// TIA Portal V19 export
FUNCTION_BLOCK "TYPIC_C215_SF_PBK"   // FB125, FBD
{ S7_Optimized_Access := 'TRUE' }
AUTHOR : OCOTECH
FAMILY : Typical
NAME : C215.804
// stored: MemoryReserve 10, SetENOAutomatically false
   VAR_INPUT
      STU_ALG_LCK_SIG { ExternalAccessible := 'False'; ExternalVisible := 'False'; ExternalWritable := 'False'} : USInt;   // Onderdruk alarmen
   END_VAR
   VAR_IN_OUT
      VAR_IF_PBK : "C215_VAR_IF_PBK_TYPIC";   // Struct met alle variabelen ontvangen van de functie (IF) in de interne sturing van het intern verlicht pictogram kopdeur
   END_VAR
   VAR
      SIG { ExternalWritable := 'False'} : Struct   // Signaleringen
         AA01 : Bool;   // Intern verlicht pictogram kopdeur niet observeerbaar
         AA02 : Bool;   // Algemene storing
         A001 : Bool;   // Beveiliging aangesproken
         A002 : Bool;   // Storing batterij
      END_STRUCT;
      VAR { ExternalWritable := 'False'} : Struct   // Variabelen
         OBS : USInt;   // Observeerbaarheid
         RNO : USInt;   // Reden niet observeerbaar
         AUT : USInt;   // Beveiliging aangesproken
         VGV_SIG_VOP : Bool;   // TRUE = Signaleringen vrijgegeven voor verkeersoperator FALSE = Onderdrukt
      END_STRUCT;
      HF_BST_OBS { ExternalAccessible := 'False'; ExternalVisible := 'False'; ExternalWritable := 'False'} : "TYPIC_HF_BST_OBS";   // Hulp functie besturing
   END_VAR
BEGIN
END_FUNCTION_BLOCK
